(* PLC project Senza_nome, Sconosciuto Senza_nome 1 *)
(* stored: creationDateTime 2024-07-29T17:39:24, modificationDateTime 2024-07-30T08:59:42 *)

FUNCTION_BLOCK LE_0
  VAR_INPUT
    IN1 : INT;
    IN2 : INT;
  END_VAR
  VAR_OUTPUT
    OUT : BOOL;
  END_VAR
  VAR
    i : INT;
  END_VAR

            OUT:=FALSE;
if IN1 <= IN2 THEN
  OUT :=TRUE;
end_if;
i:=0;
if IN1 = 12 then
  while i<4 do
    OUT:=FALSE;
  end_while;
 end_if;   
          
END_FUNCTION_BLOCK

FUNCTION_BLOCK stop_cycle
  VAR_OUTPUT
    OUT_MV1 : BOOL;
    OUT_MV2 : BOOL;
  END_VAR

            OUT_MV1 := FALSE;
OUT_MV2 := FALSE;

          
END_FUNCTION_BLOCK

FUNCTION_BLOCK valves_handler
  VAR_INPUT
    IN1 : INT;
    IN_TLB1 : INT;
    IN_TLB2 : INT;
  END_VAR
  VAR_OUTPUT
    OUT_MV1 : BOOL;
    OUT_MV2 : BOOL;
  END_VAR
  VAR
    real_value : INT;
  END_VAR

            
real_value :=  IN1 - 5;

if real_value <= IN_TLB2 then
  OUT_MV2 := FALSE;
  OUT_MV1 := TRUE;
end_if;

if real_value >= IN_TLB1 THEN
  OUT_MV2 := TRUE;
  OUT_MV1 := FALSE;
end_if;



          
END_FUNCTION_BLOCK

PROGRAM program0
  VAR_INPUT
    TLB2 : INT;
    TLB1 : INT;
    STOP : BOOL;
    START : BOOL;
    IN1 : INT;
    VALUE : INT;
  END_VAR
  VAR_OUTPUT
    MV1 : BOOL;
    MV2 : BOOL;
    CYCLE_ON : BOOL;
  END_VAR
  VAR
    stop_cycle0 : stop_cycle;
    valves_handler0 : valves_handler;
    LE_00 : LE_0;
  END_VAR

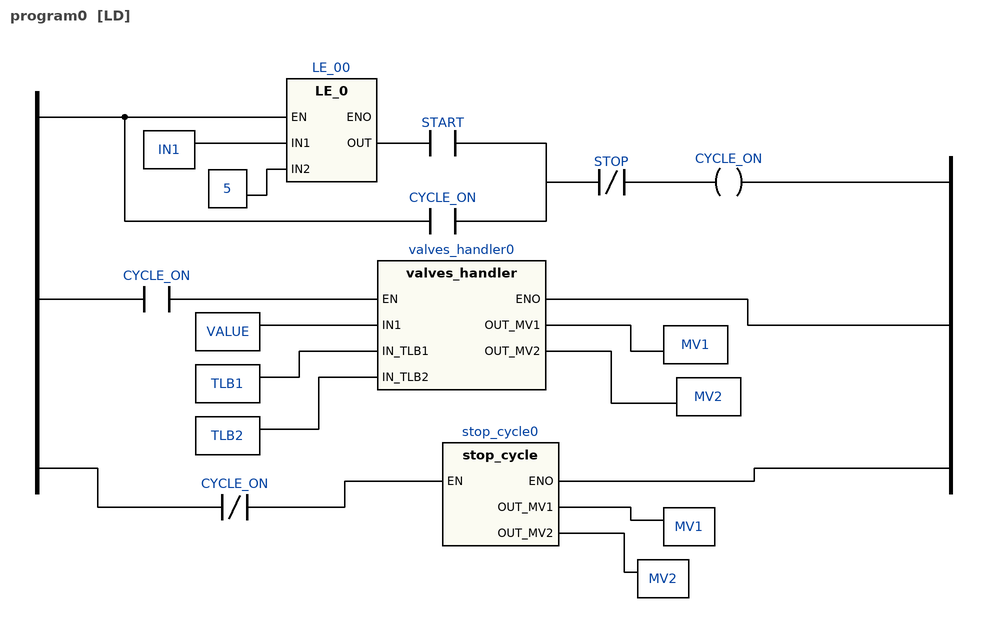
(* LD diagram, written out as Structured Text *)
valves_handler0(EN := CYCLE_ON, IN1 := VALUE, IN_TLB1 := TLB1, IN_TLB2 := TLB2);
IF valves_handler0.ENO THEN MV1 := valves_handler0.OUT_MV1; END_IF;
IF valves_handler0.ENO THEN MV2 := valves_handler0.OUT_MV2; END_IF;
LE_00(IN1 := IN1, IN2 := 5);
CYCLE_ON := (CYCLE_ON OR LE_00.OUT AND START) AND NOT STOP;
stop_cycle0(EN := NOT CYCLE_ON);
IF stop_cycle0.ENO THEN MV1 := stop_cycle0.OUT_MV1; END_IF;
IF stop_cycle0.ENO THEN MV2 := stop_cycle0.OUT_MV2; END_IF;
END_PROGRAM

CONFIGURATION Config0
  RESOURCE Res0 ON PLC
    TASK task0(INTERVAL := T#20ms, PRIORITY := 0);
    PROGRAM instance0 WITH task0 : program0;
  END_RESOURCE
END_CONFIGURATION
